// TIA Portal V18 export
DATA_BLOCK "_MAIN_DB"   // DB53
{ S7_Optimized_Access := 'TRUE' }
VERSION : 0.1
// stored: AutoNumber true, DBAccessibleFromOPCUA true, IsOnlyStoredInLoadMemory false, IsRetainMemResEnabled false, IsWriteProtectedInAS false, MemoryReserve 100
   VAR
      CLOCK_S_P_SCAN { ExternalWritable := 'False'; S7_SetPoint := 'True'} : Real := 0.03;
      AllModulesLive : Bool;
      сервисный_ключ : Bool := FALSE;
      медленно : Bool;
      bDefectsReset : Bool;
      bGoToDefectNow : Bool;
      GoToSpotNow : Bool;
      DefectsAllFound_beepResetMe : Bool;
      cycleDoneResetMe : Bool;
      Mot_Targets { S7_SetPoint := 'True'} : "typePositions";
      Mot_Positions { S7_SetPoint := 'True'} : "typePositions";
      MotCalibaratedAr { ExternalWritable := 'False'; S7_SetPoint := 'True'} : "typeGuideAxisBool";
      MotAllCalibrated { ExternalWritable := 'False'; S7_SetPoint := 'True'} : Bool;
      MotArrived { S7_SetPoint := 'True'} : "typeGuideAxisBool";
      MotAllArrived : Bool;
      desk_xAny : Bool;
      buz_alarm_er_count_change : Bool;
      buz_alarm_doorsClosedOpen : Bool;
   END_VAR
   VAR RETAIN
      главный_пульт_медлен : Bool;
   END_VAR
   VAR
      v_auto : Real := 110.0;
      Static_1 : Real := 50.0;
   END_VAR
BEGIN
END_DATA_BLOCK
